Staubli VAL3: getPoint.pgx

public program getPoint(string& x_sPoint)
begin
  //
  x_sPoint=sPointName
end
